TYPE E_AnalysisIDs :
(
	(* analysis chain *)
	eID_Source := 1,
	eID_MagSpec,
	eID_PowSpec,
	eID_SinkMag,
	eID_SinkPow
	//eID_Spectrum,
	//eID_Sink
	
) UDINT;
END_TYPE

(* stored: Version 1.1.0.1, ProductVersion 3.1.4024.3
   DUT E_AnalysisIDs: Id {986ef521-a979-48e2-815b-4873c48699c5} *)
